PROGRAM MAIN
VAR
	bDoOnce : bool := true;
END_VAR

IF bDoOnce THEN
	bDoOnce := FALSE;
	P_ADSCommManager.FB_init(FALSE,FALSE);
END_IF
P_MQTT_Agent();
P_DatabaseExchange();
//P_DBTest();
P_ADSCommManager();

END_PROGRAM

(* stored: Version 1.1.0.1, ProductVersion 3.1.4024.9
   POU MAIN: Id {9090ab64-2610-4d43-b7e3-1a5c7b9c4749}, SpecialFunc None *)
